Fanuc TP program (LS listing): ground_truth.ls

/PROG  TOR_XL_LEARN_V7
/ATTR
OWNER		= MNEDITOR;
COMMENT		= "WeldPRO Auto-Gen";
PROG_SIZE	= 7125;
CREATE		= DATE 26-07-31  TIME 10:12:18;
MODIFIED	= DATE 26-07-31  TIME 11:17:00;
FILE_NAME	= TOR_XL_L;
VERSION		= 0;
LINE_COUNT	= 113;
MEMORY_SIZE	= 7445;
PROTECT		= READ_WRITE;
TCD:  STACK_SIZE	= 0,
      TASK_PRIORITY	= 50,
      TIME_SLICE	= 0,
      BUSY_LAMP_OFF	= 0,
      ABORT_REQUEST	= 0,
      PAUSE_REQUEST	= 0;
DEFAULT_GROUP	= 1,*,*,*,*;
CONTROL_CODE	= 00000000 00000000;
/APPL
/MN
   1:  !WeldPRO Auto-Generated TPP ;
   2:  !TOR_XL_2026, TOR_xl_2907 ;
   3:   ;
   4:  UFRAME_NUM=2 ;
   5:  UTOOL_NUM=2 ;
   6:  !Feature Approach ;
   7:J P[1]{
   GP1:
	UF : 2, UT : 2,		CONFIG : 'F D T, 0, 0, 0',
	X =   924.335  mm,	Y =   780.986  mm,	Z =  -268.284  mm,
	W =  -106.495 deg,	P =   -15.000 deg,	R =    94.234 deg
};
P[2]{
   GP1:
	UF : 2, UT : 2,		CONFIG : 'F D T, 0, 0, 0',
	X =  1022.235  mm,	Y =   779.798  mm,	Z =  -236.737  mm,
	W =  -106.501 deg,	P =   -14.998 deg,	R =    94.232 deg
};
P[3]{
   GP1:
	UF : 2, UT : 2,		CONFIG : 'F D T, 0, 0, 0',
	X =  1022.568  mm,	Y =   797.695  mm,	Z =  -237.522  mm,
	W =  -106.481 deg,	P =   -15.218 deg,	R =    85.605 deg
};
P[4]{
   GP1:
	UF : 2, UT : 2,		CONFIG : 'F D T, 0, 0, 0',
	X =  1023.701  mm,	Y =   807.403  mm,	Z =  -237.378  mm,
	W =  -106.456 deg,	P =   -15.335 deg,	R =    80.815 deg
};
P[5]{
   GP1:
	UF : 2, UT : 2,		CONFIG : 'F D T, 0, 0, 0',
	X =  1025.632  mm,	Y =   817.115  mm,	Z =  -237.774  mm,
	W =  -106.423 deg,	P =   -15.449 deg,	R =    76.083 deg
};
P[6]{
   GP1:
	UF : 2, UT : 2,		CONFIG : 'F D T, 0, 0, 0',
	X =  1028.723  mm,	Y =   826.479  mm,	Z =  -237.900  mm,
	W =  -106.378 deg,	P =   -15.565 deg,	R =    71.217 deg
};
P[7]{
   GP1:
	UF : 2, UT : 2,		CONFIG : 'F D T, 0, 0, 0',
	X =  1032.825  mm,	Y =   835.377  mm,	Z =  -238.058  mm,
	W =  -106.322 deg,	P =   -15.679 deg,	R =    66.207 deg
};
P[8]{
   GP1:
	UF : 2, UT : 2,		CONFIG : 'F D T, 0, 0, 0',
	X =  1037.316  mm,	Y =   843.891  mm,	Z =  -237.866  mm,
	W =  -106.254 deg,	P =   -15.791 deg,	R =    61.015 deg
};
P[9]{
   GP1:
	UF : 2, UT : 2,		CONFIG : 'F D T, 0, 0, 0',
	X =  1042.313  mm,	Y =   852.241  mm,	Z =  -238.080  mm,
	W =  -106.177 deg,	P =   -15.894 deg,	R =    55.979 deg
};
P[10]{
   GP1:
	UF : 2, UT : 2,		CONFIG : 'F D T, 0, 0, 0',
	X =  1047.939  mm,	Y =   860.013  mm,	Z =  -237.764  mm,
	W =  -106.096 deg,	P =   -15.986 deg,	R =    51.162 deg
};
P[11]{
   GP1:
	UF : 2, UT : 2,		CONFIG : 'F D T, 0, 0, 0',
	X =  1054.535  mm,	Y =   867.095  mm,	Z =  -237.746  mm,
	W =  -106.012 deg,	P =   -16.066 deg,	R =    46.632 deg
};
P[12]{
   GP1:
	UF : 2, UT : 2,		CONFIG : 'F D T, 0, 0, 0',
	X =  1061.438  mm,	Y =   873.876  mm,	Z =  -237.867  mm,
	W =  -105.919 deg,	P =   -16.142 deg,	R =    41.952 deg
};
P[13]{
   GP1:
	UF : 2, UT : 2,		CONFIG : 'F D T, 0, 0, 0',
	X =  1068.971  mm,	Y =   880.167  mm,	Z =  -237.773  mm,
	W =  -105.870 deg,	P =   -16.177 deg,	R =    39.609 deg
};
P[14]{
   GP1:
	UF : 2, UT : 2,		CONFIG : 'F D T, 0, 0, 0',
	X =  1076.532  mm,	Y =   886.144  mm,	Z =  -237.673  mm,
	W =  -105.777 deg,	P =   -16.235 deg,	R =    35.365 deg
};
P[15]{
   GP1:
	UF : 2, UT : 2,		CONFIG : 'F D T, 0, 0, 0',
	X =  1084.991  mm,	Y =   890.765  mm,	Z =  -237.610  mm,
	W =  -105.677 deg,	P =   -16.289 deg,	R =    30.964 deg
};
P[16]{
   GP1:
	UF : 2, UT : 2,		CONFIG : 'F D T, 0, 0, 0',
	X =  1093.376  mm,	Y =   895.601  mm,	Z =  -237.769  mm,
	W =  -105.579 deg,	P =   -16.333 deg,	R =    26.830 deg
};
P[17]{
   GP1:
	UF : 2, UT : 2,		CONFIG : 'F D T, 0, 0, 0',
	X =  1101.872  mm,	Y =   899.866  mm,	Z =  -236.675  mm,
	W =  -105.536 deg,	P =   -16.344 deg,	R =    25.018 deg
};
P[18]{
   GP1:
	UF : 2, UT : 2,		CONFIG : 'F D T, 0, 0, 0',
	X =  1111.490  mm,	Y =   904.234  mm,	Z =  -236.698  mm,
	W =  -116.027 deg,	P =   -16.063 deg,	R =    30.267 deg
};
P[19]{
   GP1:
	UF : 2, UT : 2,		CONFIG : 'F D T, 0, 0, 0',
	X =  1119.627  mm,	Y =   907.760  mm,	Z =  -233.296  mm,
	W =  -126.877 deg,	P =   -15.356 deg,	R =    25.893 deg
};
P[20]{
   GP1:
	UF : 2, UT : 2,		CONFIG : 'F D T, 0, 0, 0',
	X =  1124.960  mm,	Y =   911.183  mm,	Z =  -228.098  mm,
	W =  -119.393 deg,	P =   -15.981 deg,	R =    16.221 deg
};
P[21]{
   GP1:
	UF : 2, UT : 2,		CONFIG : 'F D T, 0, 0, 0',
	X =  1130.296  mm,	Y =   915.061  mm,	Z =  -221.386  mm,
	W =  -115.329 deg,	P =   -16.208 deg,	R =    11.788 deg
};
P[22]{
   GP1:
	UF : 2, UT : 2,		CONFIG : 'F D T, 0, 0, 0',
	X =  1136.174  mm,	Y =   916.745  mm,	Z =  -213.688  mm,
	W =  -112.639 deg,	P =   -16.315 deg,	R =     9.714 deg
};
P[23]{
   GP1:
	UF : 2, UT : 2,		CONFIG : 'F D T, 0, 0, 0',
	X =  1143.006  mm,	Y =   918.720  mm,	Z =  -205.948  mm,
	W =  -110.015 deg,	P =   -16.386 deg,	R =     9.649 deg
};
P[24]{
   GP1:
	UF : 2, UT : 2,		CONFIG : 'F D T, 0, 0, 0',
	X =  1147.522  mm,	Y =   919.314  mm,	Z =  -202.449  mm,
	W =  -108.552 deg,	P =   -16.418 deg,	R =     8.950 deg
};
P[25]{
   GP1:
	UF : 2, UT : 2,		CONFIG : 'F D T, 0, 0, 0',
	X =  1160.792  mm,	Y =   921.083  mm,	Z =  -198.283  mm,
	W =  -105.409 deg,	P =   -16.443 deg,	R =     6.805 deg
};
P[26]{
   GP1:
	UF : 2, UT : 2,		CONFIG : 'F D T, 0, 0, 0',
	X =  1170.470  mm,	Y =   922.681  mm,	Z =  -197.886  mm,
	W =  -104.866 deg,	P =   -16.444 deg,	R =     5.597 deg
};
P[27]{
   GP1:
	UF : 2, UT : 2,		CONFIG : 'F D T, 0, 0, 0',
	X =  1180.180  mm,	Y =   922.877  mm,	Z =  -197.815  mm,
	W =  -104.887 deg,	P =   -16.444 deg,	R =     3.523 deg
};
P[28]{
   GP1:
	UF : 2, UT : 2,		CONFIG : 'F D T, 0, 0, 0',
	X =  1189.472  mm,	Y =   923.271  mm,	Z =  -197.392  mm,
	W =  -104.930 deg,	P =   -16.439 deg,	R =     -.729 deg
};
P[29]{
   GP1:
	UF : 2, UT : 2,		CONFIG : 'F D T, 0, 0, 0',
	X =  1198.710  mm,	Y =   922.735  mm,	Z =  -197.052  mm,
	W =  -104.979 deg,	P =   -16.424 deg,	R =    -5.541 deg
};
P[30]{
   GP1:
	UF : 2, UT : 2,		CONFIG : 'F D T, 0, 0, 0',
	X =  1207.948  mm,	Y =   921.183  mm,	Z =  -197.083  mm,
	W =  -105.028 deg,	P =   -16.400 deg,	R =   -10.259 deg
};
P[31]{
   GP1:
	UF : 2, UT : 2,		CONFIG : 'F D T, 0, 0, 0',
	X =  1217.269  mm,	Y =   919.559  mm,	Z =  -197.318  mm,
	W =  -105.070 deg,	P =   -16.371 deg,	R =   -14.490 deg
};
P[32]{
   GP1:
	UF : 2, UT : 2,		CONFIG : 'F D T, 0, 0, 0',
	X =  1226.213  mm,	Y =   916.470  mm,	Z =  -197.180  mm,
	W =  -105.112 deg,	P =   -16.334 deg,	R =   -18.515 deg
};
P[33]{
   GP1:
	UF : 2, UT : 2,		CONFIG : 'F D T, 0, 0, 0',
	X =  1235.315  mm,	Y =   914.048  mm,	Z =  -197.074  mm,
	W =  -105.158 deg,	P =   -16.285 deg,	R =   -23.051 deg
};
P[34]{
   GP1:
	UF : 2, UT : 2,		CONFIG : 'F D T, 0, 0, 0',
	X =  1243.302  mm,	Y =   909.677  mm,	Z =  -196.746  mm,
	W =  -105.219 deg,	P =   -16.204 deg,	R =   -29.417 deg
};
P[35]{
   GP1:
	UF : 2, UT : 2,		CONFIG : 'F D T, 0, 0, 0',
	X =  1258.182  mm,	Y =   898.503  mm,	Z =  -196.412  mm,
	W =  -105.307 deg,	P =   -16.055 deg,	R =   -38.974 deg
};
P[36]{
   GP1:
	UF : 2, UT : 2,		CONFIG : 'F D T, 0, 0, 0',
	X =  1265.960  mm,	Y =   892.307  mm,	Z =  -196.261  mm,
	W =  -105.302 deg,	P =   -16.063 deg,	R =   -38.625 deg
};
P[37]{
   GP1:
	UF : 2, UT : 2,		CONFIG : 'F D T, 0, 0, 0',
	X =  1273.236  mm,	Y =   886.609  mm,	Z =  -196.399  mm,
	W =  -105.469 deg,	P =   -15.944 deg,	R =   -44.976 deg
};
P[38]{
   GP1:
	UF : 2, UT : 2,		CONFIG : 'F D T, 0, 0, 0',
	X =  1280.282  mm,	Y =   880.166  mm,	Z =  -196.589  mm,
	W =  -105.661 deg,	P =   -15.890 deg,	R =   -47.714 deg
};
P[39]{
   GP1:
	UF : 2, UT : 2,		CONFIG : 'F D T, 0, 0, 0',
	X =  1286.214  mm,	Y =   873.069  mm,	Z =  -197.097  mm,
	W =  -106.210 deg,	P =   -15.792 deg,	R =   -52.259 deg
};
P[40]{
   GP1:
	UF : 2, UT : 2,		CONFIG : 'F D T, 0, 0, 0',
	X =  1291.960  mm,	Y =   865.636  mm,	Z =  -198.493  mm,
	W =  -106.927 deg,	P =   -15.688 deg,	R =   -56.663 deg
};
P[41]{
   GP1:
	UF : 2, UT : 2,		CONFIG : 'F D T, 0, 0, 0',
	X =  1298.125  mm,	Y =   858.485  mm,	Z =  -199.458  mm,
	W =  -107.603 deg,	P =   -15.597 deg,	R =   -60.243 deg
};
P[42]{
   GP1:
	UF : 2, UT : 2,		CONFIG : 'F D T, 0, 0, 0',
	X =  1302.313  mm,	Y =   850.066  mm,	Z =  -200.700  mm,
	W =  -108.271 deg,	P =   -15.504 deg,	R =   -63.685 deg
};
P[43]{
   GP1:
	UF : 2, UT : 2,		CONFIG : 'F D T, 0, 0, 0',
	X =  1306.418  mm,	Y =   841.496  mm,	Z =  -202.616  mm,
	W =  -109.143 deg,	P =   -15.377 deg,	R =   -68.203 deg
};
P[44]{
   GP1:
	UF : 2, UT : 2,		CONFIG : 'F D T, 0, 0, 0',
	X =  1309.626  mm,	Y =   832.636  mm,	Z =  -203.983  mm,
	W =  -109.899 deg,	P =   -15.253 deg,	R =   -72.505 deg
};
P[45]{
   GP1:
	UF : 2, UT : 2,		CONFIG : 'F D T, 0, 0, 0',
	X =  1313.991  mm,	Y =   823.756  mm,	Z =  -205.543  mm,
	W =  -110.273 deg,	P =   -15.181 deg,	R =   -74.981 deg
};
P[46]{
   GP1:
	UF : 2, UT : 2,		CONFIG : 'F D T, 0, 0, 0',
	X =  1315.648  mm,	Y =   814.078  mm,	Z =  -206.560  mm,
	W =  -110.635 deg,	P =   -14.305 deg,	R =   -78.232 deg
};
P[47]{
   GP1:
	UF : 2, UT : 2,		CONFIG : 'F D T, 0, 0, 0',
	X =  1317.405  mm,	Y =   804.547  mm,	Z =  -207.700  mm,
	W =  -111.054 deg,	P =   -14.769 deg,	R =   -83.164 deg
};
P[48]{
   GP1:
	UF : 2, UT : 2,		CONFIG : 'F D T, 0, 0, 0',
	X =  1318.647  mm,	Y =   795.054  mm,	Z =  -207.740  mm,
	W =  -111.190 deg,	P =   -15.305 deg,	R =   -88.308 deg
};
P[49]{
   GP1:
	UF : 2, UT : 2,		CONFIG : 'F D T, 0, 0, 0',
	X =  1318.199  mm,	Y =   785.251  mm,	Z =  -207.675  mm,
	W =  -111.129 deg,	P =   -15.645 deg,	R =   -91.614 deg
};
P[50]{
   GP1:
	UF : 2, UT : 2,		CONFIG : 'F D T, 0, 0, 0',
	X =  1318.191  mm,	Y =   775.248  mm,	Z =  -207.453  mm,
	W =  -110.757 deg,	P =   -14.624 deg,	R =   -96.575 deg
};
P[51]{
   GP1:
	UF : 2, UT : 2,		CONFIG : 'F D T, 0, 0, 0',
	X =  1317.011  mm,	Y =   765.561  mm,	Z =  -206.391  mm,
	W =  -110.276 deg,	P =   -14.535 deg,	R =  -100.836 deg
};
P[52]{
   GP1:
	UF : 2, UT : 2,		CONFIG : 'F D T, 0, 0, 0',
	X =  1314.771  mm,	Y =   756.233  mm,	Z =  -204.510  mm,
	W =  -109.635 deg,	P =   -14.447 deg,	R =  -105.265 deg
};
P[53]{
   GP1:
	UF : 2, UT : 2,		CONFIG : 'F D T, 0, 0, 0',
	X =  1312.721  mm,	Y =   746.667  mm,	Z =  -202.940  mm,
	W =  -109.083 deg,	P =   -14.382 deg,	R =  -108.625 deg
};
P[54]{
   GP1:
	UF : 2, UT : 2,		CONFIG : 'F D T, 0, 0, 0',
	X =  1309.267  mm,	Y =   737.584  mm,	Z =  -201.271  mm,
	W =  -108.349 deg,	P =   -14.302 deg,	R =  -112.873 deg
};
P[55]{
   GP1:
	UF : 2, UT : 2,		CONFIG : 'F D T, 0, 0, 0',
	X =  1305.247  mm,	Y =   728.759  mm,	Z =  -199.319  mm,
	W =  -107.748 deg,	P =   -14.239 deg,	R =  -116.265 deg
};
P[56]{
   GP1:
	UF : 2, UT : 2,		CONFIG : 'F D T, 0, 0, 0',
	X =  1301.204  mm,	Y =   719.910  mm,	Z =  -197.748  mm,
	W =  -106.924 deg,	P =   -14.148 deg,	R =  -121.191 deg
};
P[57]{
   GP1:
	UF : 2, UT : 2,		CONFIG : 'F D T, 0, 0, 0',
	X =  1295.838  mm,	Y =   711.862  mm,	Z =  -196.064  mm,
	W =  -106.269 deg,	P =   -14.066 deg,	R =  -125.698 deg
};
P[58]{
   GP1:
	UF : 2, UT : 2,		CONFIG : 'F D T, 0, 0, 0',
	X =  1290.543  mm,	Y =   703.652  mm,	Z =  -194.640  mm,
	W =  -105.781 deg,	P =   -13.988 deg,	R =  -130.143 deg
};
P[59]{
   GP1:
	UF : 2, UT : 2,		CONFIG : 'F D T, 0, 0, 0',
	X =  1284.308  mm,	Y =   696.148  mm,	Z =  -193.200  mm,
	W =  -105.527 deg,	P =   -13.913 deg,	R =  -134.519 deg
};
P[60]{
   GP1:
	UF : 2, UT : 2,		CONFIG : 'F D T, 0, 0, 0',
	X =  1277.409  mm,	Y =   688.928  mm,	Z =  -193.391  mm,
	W =  -105.437 deg,	P =   -13.849 deg,	R =  -138.629 deg
};
P[61]{
   GP1:
	UF : 2, UT : 2,		CONFIG : 'F D T, 0, 0, 0',
	X =  1270.207  mm,	Y =   682.034  mm,	Z =  -193.209  mm,
	W =  -105.429 deg,	P =   -13.831 deg,	R =  -139.837 deg
};
P[62]{
   GP1:
	UF : 2, UT : 2,		CONFIG : 'F D T, 0, 0, 0',
	X =  1262.946  mm,	Y =   675.226  mm,	Z =  -192.927  mm,
	W =  -105.443 deg,	P =   -13.863 deg,	R =  -137.727 deg
};
P[63]{
   GP1:
	UF : 2, UT : 2,		CONFIG : 'F D T, 0, 0, 0',
	X =  1255.283  mm,	Y =   668.864  mm,	Z =  -192.727  mm,
	W =  -105.373 deg,	P =   -13.729 deg,	R =  -147.436 deg
};
P[64]{
   GP1:
	UF : 2, UT : 2,		CONFIG : 'F D T, 0, 0, 0',
	X =  1246.960  mm,	Y =   662.961  mm,	Z =  -193.056  mm,
	W =  -105.298 deg,	P =   -13.637 deg,	R =  -156.529 deg
};
P[65]{
   GP1:
	UF : 2, UT : 2,		CONFIG : 'F D T, 0, 0, 0',
	X =  1237.849  mm,	Y =   658.778  mm,	Z =  -192.988  mm,
	W =  -105.277 deg,	P =   -13.618 deg,	R =  -158.976 deg
};
P[66]{
   GP1:
	UF : 2, UT : 2,		CONFIG : 'F D T, 0, 0, 0',
	X =  1228.397  mm,	Y =   655.398  mm,	Z =  -192.898  mm,
	W =  -105.241 deg,	P =   -13.592 deg,	R =  -162.969 deg
};
P[67]{
   GP1:
	UF : 2, UT : 2,		CONFIG : 'F D T, 0, 0, 0',
	X =  1218.855  mm,	Y =   652.630  mm,	Z =  -192.382  mm,
	W =  -105.203 deg,	P =   -13.573 deg,	R =  -167.022 deg
};
P[68]{
   GP1:
	UF : 2, UT : 2,		CONFIG : 'F D T, 0, 0, 0',
	X =  1209.028  mm,	Y =   649.276  mm,	Z =  -193.088  mm,
	W =  -105.159 deg,	P =   -13.560 deg,	R =  -171.569 deg
};
P[69]{
   GP1:
	UF : 2, UT : 2,		CONFIG : 'F D T, 0, 0, 0',
	X =  1199.001  mm,	Y =   649.480  mm,	Z =  -192.484  mm,
	W =  -105.113 deg,	P =   -13.556 deg,	R =  -176.312 deg
};
P[70]{
   GP1:
	UF : 2, UT : 2,		CONFIG : 'F D T, 0, 0, 0',
	X =  1189.000  mm,	Y =   649.734  mm,	Z =  -192.404  mm,
	W =  -105.068 deg,	P =   -13.561 deg,	R =   179.213 deg
};
P[71]{
   GP1:
	UF : 2, UT : 2,		CONFIG : 'F D T, 0, 0, 0',
	X =  1178.909  mm,	Y =   649.471  mm,	Z =  -192.642  mm,
	W =  -105.038 deg,	P =   -13.569 deg,	R =   176.231 deg
};
P[72]{
   GP1:
	UF : 2, UT : 2,		CONFIG : 'F D T, 0, 0, 0',
	X =  1168.932  mm,	Y =   650.575  mm,	Z =  -192.753  mm,
	W =  -105.207 deg,	P =   -13.572 deg,	R =   175.290 deg
};
P[73]{
   GP1:
	UF : 2, UT : 2,		CONFIG : 'F D T, 0, 0, 0',
	X =  1159.347  mm,	Y =   651.353  mm,	Z =  -193.648  mm,
	W =  -107.012 deg,	P =   -13.569 deg,	R =   174.537 deg
};
P[74]{
   GP1:
	UF : 2, UT : 2,		CONFIG : 'F D T, 0, 0, 0',
	X =  1150.400  mm,	Y =   651.622  mm,	Z =  -197.184  mm,
	W =  -109.414 deg,	P =   -13.538 deg,	R =   174.483 deg
};
P[75]{
   GP1:
	UF : 2, UT : 2,		CONFIG : 'F D T, 0, 0, 0',
	X =  1142.832  mm,	Y =   652.900  mm,	Z =  -202.592  mm,
	W =  -112.196 deg,	P =   -13.466 deg,	R =   175.323 deg
};
P[76]{
   GP1:
	UF : 2, UT : 2,		CONFIG : 'F D T, 0, 0, 0',
	X =  1136.327  mm,	Y =   653.526  mm,	Z =  -210.688  mm,
	W =  -114.872 deg,	P =   -13.369 deg,	R =   175.422 deg
};
P[77]{
   GP1:
	UF : 2, UT : 2,		CONFIG : 'F D T, 0, 0, 0',
	X =  1129.904  mm,	Y =   655.680  mm,	Z =  -218.910  mm,
	W =  -120.114 deg,	P =   -13.109 deg,	R =   172.293 deg
};
P[78]{
   GP1:
	UF : 2, UT : 2,		CONFIG : 'F D T, 0, 0, 0',
	X =  1123.644  mm,	Y =   659.664  mm,	Z =  -226.829  mm,
	W =  -126.809 deg,	P =   -12.620 deg,	R =   167.791 deg
};
P[79]{
   GP1:
	UF : 2, UT : 2,		CONFIG : 'F D T, 0, 0, 0',
	X =  1115.564  mm,	Y =   663.921  mm,	Z =  -231.315  mm,
	W =  -119.561 deg,	P =   -13.285 deg,	R =   157.806 deg
};
P[80]{
   GP1:
	UF : 2, UT : 2,		CONFIG : 'F D T, 0, 0, 0',
	X =  1106.454  mm,	Y =   668.458  mm,	Z =  -232.994  mm,
	W =  -107.325 deg,	P =   -13.741 deg,	R =   154.437 deg
};
P[81]{
   GP1:
	UF : 2, UT : 2,		CONFIG : 'F D T, 0, 0, 0',
	X =  1097.283  mm,	Y =   672.647  mm,	Z =  -233.048  mm,
	W =  -105.746 deg,	P =   -13.749 deg,	R =   154.142 deg
};
P[82]{
   GP1:
	UF : 2, UT : 2,		CONFIG : 'F D T, 0, 0, 0',
	X =  1088.436  mm,	Y =   677.579  mm,	Z =  -233.491  mm,
	W =  -105.804 deg,	P =   -13.784 deg,	R =   151.506 deg
};
P[83]{
   GP1:
	UF : 2, UT : 2,		CONFIG : 'F D T, 0, 0, 0',
	X =  1079.959  mm,	Y =   682.860  mm,	Z =  -233.353  mm,
	W =  -105.885 deg,	P =   -13.838 deg,	R =   147.739 deg
};
P[84]{
   GP1:
	UF : 2, UT : 2,		CONFIG : 'F D T, 0, 0, 0',
	X =  1071.661  mm,	Y =   688.646  mm,	Z =  -233.745  mm,
	W =  -105.988 deg,	P =   -13.918 deg,	R =   142.681 deg
};
P[85]{
   GP1:
	UF : 2, UT : 2,		CONFIG : 'F D T, 0, 0, 0',
	X =  1063.877  mm,	Y =   695.233  mm,	Z =  -234.380  mm,
	W =  -106.084 deg,	P =   -14.001 deg,	R =   137.677 deg
};
P[86]{
   GP1:
	UF : 2, UT : 2,		CONFIG : 'F D T, 0, 0, 0',
	X =  1056.173  mm,	Y =   701.727  mm,	Z =  -234.884  mm,
	W =  -106.129 deg,	P =   -14.056 deg,	R =   135.015 deg
};
P[87]{
   GP1:
	UF : 2, UT : 2,		CONFIG : 'F D T, 0, 0, 0',
	X =  1049.454  mm,	Y =   709.307  mm,	Z =  -235.297  mm,
	W =  -106.186 deg,	P =   -14.117 deg,	R =   131.622 deg
};
P[88]{
   GP1:
	UF : 2, UT : 2,		CONFIG : 'F D T, 0, 0, 0',
	X =  1043.392  mm,	Y =   717.267  mm,	Z =  -235.532  mm,
	W =  -106.269 deg,	P =   -14.239 deg,	R =   125.999 deg
};
P[89]{
   GP1:
	UF : 2, UT : 2,		CONFIG : 'F D T, 0, 0, 0',
	X =  1037.983  mm,	Y =   725.423  mm,	Z =  -235.539  mm,
	W =  -106.343 deg,	P =   -14.367 deg,	R =   120.225 deg
};
P[90]{
   GP1:
	UF : 2, UT : 2,		CONFIG : 'F D T, 0, 0, 0',
	X =  1033.613  mm,	Y =   733.484  mm,	Z =  -235.939  mm,
	W =  -106.383 deg,	P =   -14.448 deg,	R =   116.672 deg
};
P[91]{
   GP1:
	UF : 2, UT : 2,		CONFIG : 'F D T, 0, 0, 0',
	X =  1028.796  mm,	Y =   741.302  mm,	Z =  -236.521  mm,
	W =  -106.433 deg,	P =   -14.556 deg,	R =   111.957 deg
};
P[92]{
   GP1:
	UF : 2, UT : 2,		CONFIG : 'F D T, 0, 0, 0',
	X =  1026.094  mm,	Y =   753.101  mm,	Z =  -236.440  mm,
	W =  -106.465 deg,	P =   -14.714 deg,	R =   105.666 deg
};
P[93]{
   GP1:
	UF : 2, UT : 2,		CONFIG : 'F D T, 0, 1, 0',
	X =  1022.992  mm,	Y =   762.703  mm,	Z =  -236.848  mm,
	W =  -106.480 deg,	P =   -14.798 deg,	R =   102.261 deg
};
P[94]{
   GP1:
	UF : 2, UT : 2,		CONFIG : 'F D T, 0, 1, 0',
	X =  1022.382  mm,	Y =   772.718  mm,	Z =  -237.033  mm,
	W =  -106.494 deg,	P =   -14.935 deg,	R =    96.827 deg
};
P[95]{
   GP1:
	UF : 2, UT : 2,		CONFIG : 'F D T, 0, 0, 0',
	X =  1014.789  mm,	Y =   776.665  mm,	Z =  -227.278  mm,
	W =  -106.497 deg,	P =   -14.995 deg,	R =    94.216 deg
};
P[96]{
   GP1:
	UF : 2, UT : 2,		CONFIG : 'F D T, 0, 1, 0',
	X =  1021.186  mm,	Y =   779.808  mm,	Z =  -237.142  mm,
	W =  -106.501 deg,	P =   -15.000 deg,	R =    94.236 deg
};
P[97]{
   GP1:
	UF : 2, UT : 2,		CONFIG : 'F D T, 0, 0, 0',
	X =  1021.927  mm,	Y =   787.763  mm,	Z =  -237.152  mm,
	W =  -106.492 deg,	P =   -15.098 deg,	R =    90.372 deg
};
P[98]{
   GP1:
	UF : 2, UT : 2,		CONFIG : 'F D T, 0, 1, 0',
	X =   651.995  mm,	Y =   781.694  mm,	Z =  -345.952  mm,
	W =  -106.495 deg,	P =   -15.000 deg,	R =    94.234 deg
};

/END
